// TIA Portal V21 export
TYPE "Std_stTimeStamp"
   STRUCT
      diHours { ExternalVisible := 'False'} : DInt;
      iMinutes { ExternalVisible := 'False'} : Int;
      iSeconds { ExternalVisible := 'False'} : Int;
      iMilliseconds { ExternalVisible := 'False'} : Int;
   END_STRUCT;
END_TYPE
